{attribute 'GeneratedUsingTerminal: CU2508-0000-0016'}
{attribute addProperty BoxType "CU2508-0000-0016"}
{attribute addProperty Id "InfoDataAT %I*InfoData_94A18F5E2"}
{attribute addProperty CRC "2009557638"}
{attribute addProperty Size "2"}
TYPE CU2508_77C76A86 EXTENDS EtcSlaveTerminalBase_947E5A46 :
STRUCT
	{attribute addProperty Name "InfoData"}
	InfoData : InfoData_94A18F5E;
END_STRUCT
END_TYPE

(* stored: Version 1.2.0.0, ProductVersion 3.1.4024.9
   DUT CU2508_77C76A86: Id {ffa8fd80-6049-4ec2-b940-11b1105e2408} *)
